(* IEC 61131-3 sources: horner-cscape-mcp/artifacts/projects/AddStagingAuditProject/pous, 1 file *)

(* ---- AddStagingTest.st ---- *)
PROGRAM AddStagingTest
VAR
    nVal : INT;
END_VAR
nVal := 42;
END_PROGRAM
